// TIA Portal V19 export
DATA_BLOCK "NEW OUTPUTS"   // DB70
{ S7_Optimized_Access := 'TRUE' }
// stored: MemoryReserve 100
   VAR
      "MFG FEED PUMP OP" : Bool;
      "RO 1 HPP PUMP OP" : Bool;
      "RO 2 HPP PUMP OP" : Bool;
      "CIP PUMP OP" : Bool;
      "PW TRANSFER PUMP W OP" : Bool;
      "PW TRANSFER PUMP S OP" : Bool;
      "SPARE OP1" : Bool;
      "SPARE OP2" : Bool;
      "SPARE OP3" : Bool;
      "DP-1 OP" : Bool;
      "DP-2 OP" : Bool;
      "UV-1 OP" : Bool;
      "SPARE OP4" : Bool;
      "SPARE OP5" : Bool;
      "SPARE OP6" : Bool;
      "SPARE OP7" : Bool;
      "SPARE OP8" : Bool;
      "HOOTER OP" : Bool;
      "MFG OPEN V1" : Bool;
      "MFG OPEN V2" : Bool;
      "MFG OPEN V3" : Bool;
      "MFG OPEN V4" : Bool;
      "MFG OPEN V5" : Bool;
      "MFG CLOSE V1" : Bool;
      "MFG CLOSE V2" : Bool;
      "MFG CLOSE V3" : Bool;
      "MFG CLOSE V4" : Bool;
      "MFG CLOSE V5" : Bool;
      "ACF OPEN V1" : Bool;
      "ACF OPEN V2" : Bool;
      "ACF OPEN V3" : Bool;
      "ACF OPEN V4" : Bool;
      "ACF OPEN V5" : Bool;
      "ACF CLOSE V1" : Bool;
      "ACF CLOSE V2" : Bool;
      "ACF CLOSE V3" : Bool;
      "ACF CLOSE V4" : Bool;
      "ACF CLOSE V5" : Bool;
      "SF OPEN V1" : Bool;
      "SF OPEN V2" : Bool;
      "SF OPEN V3" : Bool;
      "SF OPEN V4" : Bool;
      "SF OPEN V5" : Bool;
      "SF OPEN V6" : Bool;
      "SF OPEN V7" : Bool;
      "SF CLOSE V1" : Bool;
      "SF CLOSE V2" : Bool;
      "SF CLOSE V3" : Bool;
      "SF CLOSE V4" : Bool;
      "SF CLOSE V5" : Bool;
      "SF CLOSE V6" : Bool;
      "SF CLOSE V7" : Bool;
      "AV 1" : Bool;
      "AV 2" : Bool;
      "AV 3" : Bool;
      "AV 4" : Bool;
      "SPARE OP9" : Bool;
      "SPARE OP10" : Bool;
   END_VAR
BEGIN
END_DATA_BLOCK
